Fanuc KAREL source: kt00444.KL

-- PROVISIONAL review KL for V940-1; original PC SHA256 831edb69b5a948d46798f5ed3e4c22599dc2f2cd2ce0d7bb3aa8d8d12013f794
-- Incomplete behavior may be omitted. Consult companion uncertainty JSON. Do not deploy.
PROGRAM KT00444
%NOLOCKGROUP
VAR
  R1 : REAL
  OUT : BOOLEAN
-- UNRESOLVED_DECL H2 type=002017
BEGIN
  -- V9_ZERO_TABLE_METADATA_HINT layout=0001; no indexed target words; source/name/runtime held
  -- UNRESOLVED_PC offsets 5-16; opcodes 2E,23
  -- UNRESOLVED_PC offsets 21-35; opcodes 2E,22,9D,33,B4
  -- UNRESOLVED_PC offsets 40-63; opcodes 21,22,9D,33,B3,64,72,23
  -- UNRESOLVED_PC offsets 68-72; opcodes 7F
END KT00444
